# EPICS alarm handler configuration: alh_files/mgnt_dmp1_lgps.alhConfig
GROUP NULL LGPS:DMP1:MG01
   $COMMAND edm -x -eolc -noedit mgnt_dmp1_lgps.edl
$ALIAS LGPS
$GUIDANCE
DMP1 LGPS
   Group Name: LGPS:DMP1:MG01
   Summary PV:  LGPS:DMP1:MG01:STATSUMY
$END

GROUP LGPS:DMP1:MG01  LGPS:DMP1:1
   $COMMAND edm -x -eolc -noedit -m "DEV=LGPS:DMP1:1" mgnt_unit.edl
CHANNEL    LGPS:DMP1:1    LGPS:DMP1:1:STATMSG   -----
   $FORCEPV LGPS:DMP1:1:STATMSGSV -DATL 1 0
